// ---- VISUs/HMI_SenSimTest.TcVIS
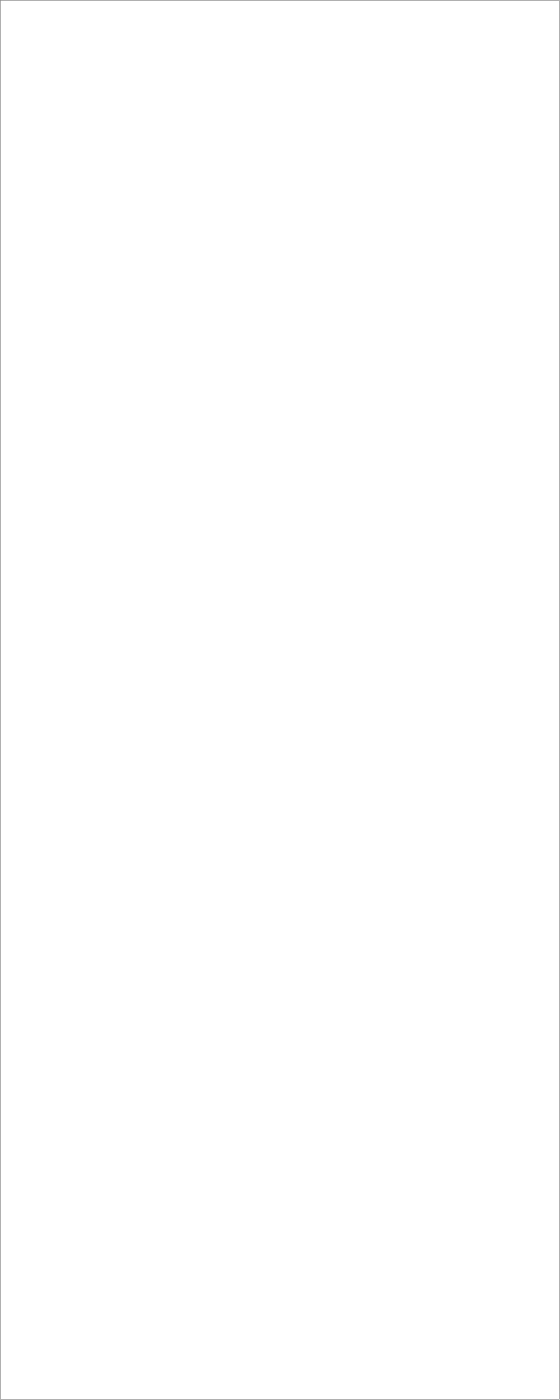
VISUALIZATION HMI_SenSimTest  // 801x2002
    Rectangle (7,175 430x823)
    Rectangle (260,175 176x823)
    Rectangle (7,875 429x23)
    Rectangle (7,741 429x23)
    Rectangle (7,174 429x23)
    Rectangle (6,16 669x143)
    Rectangle (6,17 669x32), "Manual Command Simulation From PLC"
    Checkbox (395,232 30x31), "Checkbox", tooltip "Enable Simulation", variable: stHMITIISenSimArray[iHMICbLevelSelection].bHMITIIByPassArray[1]
    ComboBoxInteger (295,235 100x25), tooltip "BackDoorSimulationMode", variable: arrTCMultiLevel[iHMICbLevelSelection].fbTCMultiLevelSeq.stMLBIO.ipAPPresentSensor, text list: 'BDList'
    RoundedRectangle (265,234 26x26), tooltip "VIO Status", colour toggle: arrTCMultiLevel[iHMICbLevelSelection].fbTCMultiLevelSeq.stMLVIO.ipAPPresentSensor
    Checkbox (263,201 164x31), "TIISen:VIOSim Override", variable: bHMIEnTIISenSimulation
    Checkbox (395,263 30x31), "Checkbox", tooltip "Enable Simulation", variable: stHMITIISenSimArray[iHMICbLevelSelection].bHMITIIByPassArray[2]
    ComboBoxInteger (295,267 100x25), tooltip "BackDoorSimulationMode", variable: arrTCMultiLevel[iHMICbLevelSelection].fbTCMultiLevelSeq.stMLBIO.ipAPPowerOn, text list: 'BDList'
    RoundedRectangle (265,265 26x26), tooltip "VIO Status", colour toggle: arrTCMultiLevel[iHMICbLevelSelection].fbTCMultiLevelSeq.stMLVIO.ipAPPowerOn
    Checkbox (395,294 30x31), "Checkbox", tooltip "Enable Simulation", variable: stHMITIISenSimArray[iHMICbLevelSelection].bHMITIIByPassArray[3]
    ComboBoxInteger (295,298 100x25), tooltip "BackDoorSimulationMode", variable: arrTCMultiLevel[iHMICbLevelSelection].fbTCMultiLevelSeq.stMLBIO.ipAPReady, text list: 'BDList'
    RoundedRectangle (265,296 26x26), tooltip "VIO Status", colour toggle: arrTCMultiLevel[iHMICbLevelSelection].fbTCMultiLevelSeq.stMLVIO.ipAPReady
    Checkbox (395,325 30x31), "Checkbox", tooltip "Enable Simulation", variable: stHMITIISenSimArray[iHMICbLevelSelection].bHMITIIByPassArray[4]
    ComboBoxInteger (295,328 100x25), tooltip "BackDoorSimulationMode", variable: arrTCMultiLevel[iHMICbLevelSelection].fbTCMultiLevelSeq.stMLBIO.ipHandlerSafeToEnterPLC, text list: 'BDList'
    RoundedRectangle (265,327 26x26), tooltip "VIO Status", colour toggle: arrTCMultiLevel[iHMICbLevelSelection].fbTCMultiLevelSeq.stMLVIO.ipHandlerSafeToEnterPLC
    Checkbox (395,356 30x31), "Checkbox", tooltip "Enable Simulation", variable: stHMITIISenSimArray[iHMICbLevelSelection].bHMITIIByPassArray[5]
    ComboBoxInteger (295,359 100x25), tooltip "BackDoorSimulationMode", variable: arrTCMultiLevel[iHMICbLevelSelection].fbTCMultiLevelSeq.stMLBIO.ipHandlerSafeToEnterHwr, text list: 'BDList'
    RoundedRectangle (265,358 26x26), tooltip "VIO Status", colour toggle: arrTCMultiLevel[iHMICbLevelSelection].fbTCMultiLevelSeq.stMLVIO.ipHandlerSafeToEnterHwr
    Checkbox (395,387 30x31), "Checkbox", tooltip "Enable Simulation", variable: stHMITIISenSimArray[iHMICbLevelSelection].bHMITIIByPassArray[6]
    ComboBoxInteger (295,390 100x25), tooltip "BackDoorSimulationMode", variable: arrTCMultiLevel[iHMICbLevelSelection].fbTCMultiLevelSeq.stMLBIO.ipCellFluidLeakage1, text list: 'BDList'
    RoundedRectangle (265,389 26x26), tooltip "VIO Status", colour toggle: arrTCMultiLevel[iHMICbLevelSelection].fbTCMultiLevelSeq.stMLVIO.ipCellFluidLeakage1
    Checkbox (395,418 30x31), "Checkbox", tooltip "Enable Simulation", variable: stHMITIISenSimArray[iHMICbLevelSelection].bHMITIIByPassArray[7]
    ComboBoxInteger (295,421 100x25), tooltip "BackDoorSimulationMode", variable: arrTCMultiLevel[iHMICbLevelSelection].fbTCMultiLevelSeq.stMLBIO.ipCellFluidLeakage2, text list: 'BDList'
    RoundedRectangle (265,420 26x26), tooltip "VIO Status", colour toggle: arrTCMultiLevel[iHMICbLevelSelection].fbTCMultiLevelSeq.stMLVIO.ipCellFluidLeakage2
    Checkbox (395,449 30x31), "Checkbox", tooltip "Enable Simulation", variable: stHMITIISenSimArray[iHMICbLevelSelection].bHMITIIByPassArray[8]
    ComboBoxInteger (295,452 100x25), tooltip "BackDoorSimulationMode", variable: arrTCMultiLevel[iHMICbLevelSelection].fbTCMultiLevelSeq.stMLBIO.ipCellGroundFault, text list: 'BDList'
    RoundedRectangle (265,451 26x26), tooltip "VIO Status", colour toggle: arrTCMultiLevel[iHMICbLevelSelection].fbTCMultiLevelSeq.stMLVIO.ipCellGroundFault
    Checkbox (395,480 30x31), "Checkbox", tooltip "Enable Simulation", variable: stHMITIISenSimArray[iHMICbLevelSelection].bHMITIIByPassArray[9]
    ComboBoxInteger (295,483 100x25), tooltip "BackDoorSimulationMode", variable: arrTCMultiLevel[iHMICbLevelSelection].fbTCMultiLevelSeq.stMLBIO.ipTesterPresent, text list: 'BDList'
    RoundedRectangle (265,482 26x26), tooltip "VIO Status", colour toggle: arrTCMultiLevel[iHMICbLevelSelection].fbTCMultiLevelSeq.stMLVIO.ipTesterPresent
    Checkbox (395,511 30x31), "Checkbox", tooltip "Enable Simulation", variable: stHMITIISenSimArray[iHMICbLevelSelection].bHMITIIByPassArray[10]
    ComboBoxInteger (295,514 100x25), tooltip "BackDoorSimulationMode", variable: arrTCMultiLevel[iHMICbLevelSelection].fbTCMultiLevelSeq.stMLBIO.ipTesterPowerOn, text list: 'BDList'
    RoundedRectangle (265,513 26x26), tooltip "VIO Status", colour toggle: arrTCMultiLevel[iHMICbLevelSelection].fbTCMultiLevelSeq.stMLVIO.ipTesterPowerOn
    Checkbox (395,542 30x31), "Checkbox", tooltip "Enable Simulation", variable: stHMITIISenSimArray[iHMICbLevelSelection].bHMITIIByPassArray[11]
    ComboBoxInteger (295,545 100x25), tooltip "BackDoorSimulationMode", variable: arrTCMultiLevel[iHMICbLevelSelection].fbTCMultiLevelSeq.stMLBIO.ipTesterReady, text list: 'BDList'
    RoundedRectangle (265,544 26x26), tooltip "VIO Status", colour toggle: arrTCMultiLevel[iHMICbLevelSelection].fbTCMultiLevelSeq.stMLVIO.ipTesterReady
    Checkbox (395,573 30x31), "Checkbox", tooltip "Enable Simulation", variable: stHMITIISenSimArray[iHMICbLevelSelection].bHMITIIByPassArray[12]
    ComboBoxInteger (295,576 100x25), tooltip "BackDoorSimulationMode", variable: arrTCMultiLevel[iHMICbLevelSelection].fbTCMultiLevelSeq.stMLBIO.ipTCCellDoorClosed, text list: 'BDList'
    RoundedRectangle (265,575 26x26), tooltip "VIO Status", colour toggle: arrTCMultiLevel[iHMICbLevelSelection].fbTCMultiLevelSeq.stMLVIO.ipTCCellDoorClosed
    Checkbox (395,604 30x31), "Checkbox", tooltip "Enable Simulation", variable: stHMITIISenSimArray[iHMICbLevelSelection].bHMITIIByPassArray[13]
    ComboBoxInteger (295,607 100x25), tooltip "BackDoorSimulationMode", variable: arrTCMultiLevel[iHMICbLevelSelection].fbTCMultiLevelSeq.stMLBIO.ipTesterLatchesClosed, text list: 'BDList'
    RoundedRectangle (265,606 26x26), tooltip "VIO Status", colour toggle: arrTCMultiLevel[iHMICbLevelSelection].fbTCMultiLevelSeq.stMLVIO.ipTesterLatchesClosed
    Checkbox (395,635 30x31), "Checkbox", tooltip "Enable Simulation", variable: stHMITIISenSimArray[iHMICbLevelSelection].bHMITIIByPassArray[14]
    ComboBoxInteger (295,638 100x25), tooltip "BackDoorSimulationMode", variable: arrTCMultiLevel[iHMICbLevelSelection].fbTCMultiLevelSeq.stMLBIO.ipTIUPresent, text list: 'BDList'
    RoundedRectangle (265,637 26x26), tooltip "VIO Status", colour toggle: arrTCMultiLevel[iHMICbLevelSelection].fbTCMultiLevelSeq.stMLVIO.ipTIUPresent
    Checkbox (395,666 30x31), "Checkbox", tooltip "Enable Simulation"
    ComboBoxInteger (295,669 100x25), tooltip "BackDoorSimulationMode", variable: arrTCMultiLevel[iHMICbLevelSelection].fbTCMultiLevelSeq.stMLBIO.ipAPPresentSensor, text list: 'BDList'
    RoundedRectangle (265,668 26x26), tooltip "VIO Status"
    Checkbox (395,697 30x31), "Checkbox", tooltip "Enable Simulation"
    ComboBoxInteger (295,700 100x25), tooltip "BackDoorSimulationMode", variable: arrTCMultiLevel[iHMICbLevelSelection].fbTCMultiLevelSeq.stMLBIO.ipAPPresentSensor, text list: 'BDList'
    RoundedRectangle (265,699 26x26), tooltip "VIO Status"
    RoundedRectangle (69,234 165x25), "01)_AP_PresentSensor*"
    Checkbox (12,232 30x31), "Checkbox", tooltip "Enable Simulation", variable: stHMITIIByPassArray[iHMICbLevelSelection].bHMITIIByPassArray[1]
    RoundedRectangle (69,265 165x25), "02)_AP_PowerOn*"
    Checkbox (12,263 30x31), "Checkbox", tooltip "Enable Simulation", variable: stHMITIIByPassArray[iHMICbLevelSelection].bHMITIIByPassArray[2]
    RoundedRectangle (69,296 165x25), "03)_AP_Ready"
    Checkbox (12,294 30x31), "Checkbox", tooltip "Enable Simulation", variable: stHMITIIByPassArray[iHMICbLevelSelection].bHMITIIByPassArray[3]
    RoundedRectangle (69,327 165x25), "04)_AP_DeactuatedPLC`*`"
    Checkbox (12,325 30x31), "Checkbox", tooltip "Enable Simulation", variable: stHMITIIByPassArray[iHMICbLevelSelection].bHMITIIByPassArray[4]
    RoundedRectangle (69,358 165x25), "05)_AP_DeactuatedHwr`*`"
    Checkbox (12,356 30x31), "Checkbox", tooltip "Enable Simulation", variable: stHMITIIByPassArray[iHMICbLevelSelection].bHMITIIByPassArray[5]
    RoundedRectangle (69,389 165x25), "06)_CellFluidLeakage1"
    Checkbox (12,387 30x31), "Checkbox", tooltip "Enable Simulation", variable: stHMITIIByPassArray[iHMICbLevelSelection].bHMITIIByPassArray[6]
    RoundedRectangle (69,420 165x25), "07)_CellFluidLeakage2"
    Checkbox (12,418 30x31), "Checkbox", tooltip "Enable Simulation", variable: stHMITIIByPassArray[iHMICbLevelSelection].bHMITIIByPassArray[7]
    RoundedRectangle (69,451 165x25), "08)_CellGroundFault"
    Checkbox (12,449 30x31), "Checkbox", tooltip "Enable Simulation", variable: stHMITIIByPassArray[iHMICbLevelSelection].bHMITIIByPassArray[8]
    RoundedRectangle (69,482 165x25), "09)_TesterPresent**"
    Checkbox (12,480 30x31), "Checkbox", tooltip "Enable Simulation", variable: stHMITIIByPassArray[iHMICbLevelSelection].bHMITIIByPassArray[9]
    RoundedRectangle (69,513 165x25), "10)_TesterPowerOn**"
    Checkbox (12,511 30x31), "Checkbox", tooltip "Enable Simulation", variable: stHMITIIByPassArray[iHMICbLevelSelection].bHMITIIByPassArray[10]
    RoundedRectangle (69,544 165x25), "11)_TesterReady"
    Checkbox (12,542 30x31), "Checkbox", tooltip "Enable Simulation", variable: stHMITIIByPassArray[iHMICbLevelSelection].bHMITIIByPassArray[11]
    RoundedRectangle (69,575 165x25), "12)_TCCellDoorClosed"
    Checkbox (12,573 30x31), "Checkbox", tooltip "Enable Simulation", variable: stHMITIIByPassArray[iHMICbLevelSelection].bHMITIIByPassArray[12]
    RoundedRectangle (69,606 165x25), "13)_TesterLatchesClosed**"
    Checkbox (12,604 30x31), "Checkbox", tooltip "Enable Simulation", variable: stHMITIIByPassArray[iHMICbLevelSelection].bHMITIIByPassArray[13]
    RoundedRectangle (69,637 165x25), "14)_TIUPresent"
    Checkbox (12,635 30x31), "Checkbox", tooltip "Enable Simulation", variable: stHMITIIByPassArray[iHMICbLevelSelection].bHMITIIByPassArray[14]
    RoundedRectangle (69,668 165x25)
    Checkbox (12,666 30x31), "Checkbox", tooltip "Enable Simulation"
    RoundedRectangle (69,699 165x25)
    Checkbox (12,697 30x31), "Checkbox", tooltip "Enable Simulation"
    Checkbox (12,202 227x31), "TII Alarm Enable Override", variable: bHMITIIBypass
    Checkbox (629,331 30x31), "Checkbox", tooltip "Enable Simulation", variable: stHMIBtnSimArray[iHMICbLevelSelection].bHMITIIByPassArray[1]
    ComboBoxInteger (483,334 140x25), tooltip "BackDoorSimulationMode", variable: arrTCMultiLevel[iHMICbLevelSelection].fbTCMultiLevelSeq.stMLBIO.ipDrawerMaintenanceModeBtn, text list: 'BDList'
    RoundedRectangle (453,333 26x26), tooltip "VIO Status", colour toggle: arrTCMultiLevel[iHMICbLevelSelection].fbTCMultiLevelSeq.stMLVIO.ipDrawerMaintenanceModeBtn
    Checkbox (629,362 30x31), "Checkbox", tooltip "Enable Simulation", variable: stHMIBtnSimArray[iHMICbLevelSelection].bHMITIIByPassArray[2]
    ComboBoxInteger (483,366 140x25), tooltip "BackDoorSimulationMode", variable: arrTCMultiLevel[iHMICbLevelSelection].fbTCMultiLevelSeq.stMLBIO.ipTCCellAbortFlowBtn, text list: 'BDList'
    RoundedRectangle (453,364 26x26), tooltip "VIO Status", colour toggle: arrTCMultiLevel[iHMICbLevelSelection].fbTCMultiLevelSeq.stMLVIO.ipTCCellAbortFlowBtn
    Checkbox (629,393 30x31), "Checkbox", tooltip "Enable Simulation", variable: stHMIBtnSimArray[iHMICbLevelSelection].bHMITIIByPassArray[3]
    ComboBoxInteger (483,397 140x25), tooltip "BackDoorSimulationMode", variable: arrTCMultiLevel[iHMICbLevelSelection].fbTCMultiLevelSeq.stMLBIO.ipTCCellDoorOpenReqBtn, text list: 'BDList'
    RoundedRectangle (453,395 26x26), tooltip "VIO Status", colour toggle: arrTCMultiLevel[iHMICbLevelSelection].fbTCMultiLevelSeq.stMLVIO.ipTCCellDoorOpenReqBtn
    Checkbox (452,300 157x31), "Btn VIO Sim Override", variable: bHMIBtnSimulation
    Checkbox (454,427 150x30), "AutoRsetEvntTrigger", variable: bHMIRsetEvntTriggerOnProductionMode
    RoundedRectangle (41,234 26x26), tooltip "VIO Status", colour toggle: ALMTC.Level[iHMICbLevelSelection].AlarmID[1]
    RoundedRectangle (41,265 26x26), tooltip "VIO Status", colour toggle: ALMTC.Level[iHMICbLevelSelection].AlarmID[2]
    RoundedRectangle (41,296 26x26), tooltip "VIO Status", colour toggle: ALMTC.Level[iHMICbLevelSelection].AlarmID[3]
    RoundedRectangle (41,327 26x26), tooltip "VIO Status", colour toggle: ALMTC.Level[iHMICbLevelSelection].AlarmID[4]
    RoundedRectangle (41,358 26x26), tooltip "VIO Status", colour toggle: ALMTC.Level[iHMICbLevelSelection].AlarmID[5]
    RoundedRectangle (41,389 26x26), tooltip "VIO Status", colour toggle: ALMTC.Level[iHMICbLevelSelection].AlarmID[6]
    RoundedRectangle (41,420 26x26), tooltip "VIO Status", colour toggle: ALMTC.Level[iHMICbLevelSelection].AlarmID[7]
    RoundedRectangle (41,451 26x26), tooltip "VIO Status", colour toggle: ALMTC.Level[iHMICbLevelSelection].AlarmID[8]
    RoundedRectangle (41,482 26x26), tooltip "VIO Status", colour toggle: ALMTC.Level[iHMICbLevelSelection].AlarmID[9]
    RoundedRectangle (41,513 26x26), tooltip "VIO Status", colour toggle: ALMTC.Level[iHMICbLevelSelection].AlarmID[10]
    RoundedRectangle (41,544 26x26), tooltip "VIO Status", colour toggle: ALMTC.Level[iHMICbLevelSelection].AlarmID[11]
    RoundedRectangle (41,575 26x26), tooltip "VIO Status", colour toggle: ALMTC.Level[iHMICbLevelSelection].AlarmID[12]
    RoundedRectangle (41,606 26x26), tooltip "VIO Status", colour toggle: ALMTC.Level[iHMICbLevelSelection].AlarmID[13]
    RoundedRectangle (41,637 26x26), tooltip "VIO Status", colour toggle: ALMTC.Level[iHMICbLevelSelection].AlarmID[14]
    RoundedRectangle (41,668 26x26), tooltip "VIO Status"
    RoundedRectangle (41,699 26x26), tooltip "VIO Status"
    Checkbox (394,766 30x31), "Checkbox", tooltip "Enable Simulation", variable: bHMIColSenSimArray[1]
    ComboBoxInteger (294,769 100x25), tooltip "BackDoorSimulationMode", variable: fbTCColumn.stTCColumnBIO.ipColumnFluid_PCW_Leakage, text list: 'BDList'
    RoundedRectangle (264,768 26x26), tooltip "VIO Status", colour toggle: fbTCColumn.stTCColumnVIO.ipColumnFluid_PCW_Leakage
    Checkbox (394,797 30x31), "Checkbox", tooltip "Enable Simulation", variable: bHMIColSenSimArray[2]
    ComboBoxInteger (294,800 100x25), tooltip "BackDoorSimulationMode", variable: fbTCColumn.stTCColumnBIO.ipAllTCDrawerRetractedinCell, text list: 'BDList'
    RoundedRectangle (264,799 26x26), tooltip "VIO Status", colour toggle: fbTCColumn.stTCColumnVIO.ipAllTCDrawerRetractedinCell
    Checkbox (394,828 30x31), "Checkbox", tooltip "Enable Simulation", variable: bHMIColSenSimArray[3]
    ComboBoxInteger (294,831 100x25), tooltip "BackDoorSimulationMode", variable: fbTCColumn.stTCColumnBIO.ipSystem_ipColumnGroundFault, text list: 'BDList'
    RoundedRectangle (264,830 26x26), tooltip "VIO Status", colour toggle: fbTCColumn.stTCColumnVIO.ipSystem_ipColumnGroundFault
    RoundedRectangle (71,769 162x25), "1)_Col_Leakage"
    Checkbox (12,767 30x31), "Checkbox", tooltip "Enable Simulation", variable: arrHMISysAlmByPass[1]
    RoundedRectangle (71,800 162x25), "2)_All_Dwr_Ret"
    Checkbox (12,799 30x31), "Checkbox", tooltip "Enable Simulation", variable: arrHMISysAlmByPass[2]
    RoundedRectangle (71,831 162x25), "3)_Col_Grd"
    Checkbox (12,830 30x31), "Checkbox", tooltip "Enable Simulation", variable: arrHMISysAlmByPass[3]
    RoundedRectangle (42,769 26x26), tooltip "VIO Status", colour toggle: ALMTC.Common.AlarmID[1]
    RoundedRectangle (42,800 26x26), tooltip "VIO Status", colour toggle: ALMTC.Common.AlarmID[2]
    RoundedRectangle (42,831 26x26), tooltip "VIO Status", colour toggle: ALMTC.Common.AlarmID[3]
    RoundedRectangle (476,233 181x25), "ButtonModeConditionSimulation"
        toggle arrHMIBtnSolidOn_Condition[iHMICbLevelSelection,iHMIBtnType]
    RoundedRectangle (449,233 25x25), colour toggle: arrHMIBtnSolidOn_Condition[iHMICbLevelSelection,iHMIBtnType]
    ComboBoxInteger (451,266 208x25), tooltip "BackDoorSimulationMode", variable: iHMIBtnType, text list: 'BtnTxtList'
    ComboBoxInteger (106,71 188x30), variable: iHMICbCmdSelection, text list: 'CmdTxtList'
    ComboBoxInteger (14,71 89x30), variable: iHMICbLevelSelection, text list: 'LevelTxtList'
    Button (12,108 281x45), "Test Command"
        tap TestManually.bTestCommand
    ComboBoxInteger (306,73 276x25), variable: TestManually.iAlarmCode, text list: 'AlarmTxtList'
    Checkbox (586,68 37x30), variable: bHMIResetAllAlarm
    Label (616,68 183x30), "Reset All"
    Label (304,50 215x30), "Individual Alarm ID:"
    Button (302,111 281x42), "Init All Level"
        tap TestManually.bInitialiseAll
    Checkbox (397,900 30x31), "Checkbox", tooltip "Enable Simulation", variable: stDebugStation.fbDBStnSeq.bTIISenSimArray[1]
    ComboBoxInteger (297,903 100x25), tooltip "BackDoorSimulationMode", variable: stDebugStation.fbDBStnSeq.stDebugStationBIO.ipDBStnAPPresentSensor, text list: 'BDList'
    RoundedRectangle (267,902 26x26), tooltip "VIO Status", colour toggle: stDebugStation.fbDBStnSeq.stDebugStationVIO.ipDBStnAPPresentSensor
    Checkbox (397,931 30x31), "Checkbox", tooltip "Enable Simulation", variable: stDebugStation.fbDBStnSeq.bTIISenSimArray[2]
    ComboBoxInteger (297,935 100x25), tooltip "BackDoorSimulationMode", variable: stDebugStation.fbDBStnSeq.stDebugStationBIO.ipDBStnAPPowerOn, text list: 'BDList'
    RoundedRectangle (267,933 26x26), tooltip "VIO Status", colour toggle: stDebugStation.fbDBStnSeq.stDebugStationVIO.ipDBStnAPPowerOn
    Checkbox (397,962 30x31), "Checkbox", tooltip "Enable Simulation", variable: stDebugStation.fbDBStnSeq.bTIISenSimArray[3]
    ComboBoxInteger (297,966 100x25), tooltip "BackDoorSimulationMode", variable: stDebugStation.fbDBStnSeq.stDebugStationBIO.ipDBStnAPReady, text list: 'BDList'
    RoundedRectangle (267,964 26x26), tooltip "VIO Status", colour toggle: stDebugStation.fbDBStnSeq.stDebugStationVIO.ipDBStnAPReady
    RoundedRectangle (71,902 165x25), "01)_AP_PresentSensor"
    Checkbox (14,900 30x31), "Checkbox", tooltip "Enable Simulation", variable: stHMITIIByPassArray[iHMICbLevelSelection].bHMITIIByPassArray[1]
    RoundedRectangle (71,933 165x25), "02)_AP_PowerOn"
    Checkbox (14,931 30x31), "Checkbox", tooltip "Enable Simulation", variable: stHMITIIByPassArray[iHMICbLevelSelection].bHMITIIByPassArray[2]
    RoundedRectangle (71,964 165x25), "03)_AP_Ready"
    Checkbox (14,962 30x31), "Checkbox", tooltip "Enable Simulation", variable: stHMITIIByPassArray[iHMICbLevelSelection].bHMITIIByPassArray[3]
    RoundedRectangle (43,902 26x26), tooltip "VIO Status", colour toggle: ALMTC.Level[iHMICbLevelSelection].AlarmID[1]
    RoundedRectangle (43,933 26x26), tooltip "VIO Status", colour toggle: ALMTC.Level[iHMICbLevelSelection].AlarmID[2]
    RoundedRectangle (43,964 26x26), tooltip "VIO Status", colour toggle: ALMTC.Level[iHMICbLevelSelection].AlarmID[3]
    Label (20,871 183x30), "DEBUG STATION"
    Label (15,171 183x30), "CELL STACK"
    Label (20,740 183x30), "COLUMN"
    Group (452,468 225x262)
        Rectangle (0,0 215x259)
        Rectangle (0,237 215x22)
        RoundedRectangle (7,206 60x26), "Level[1]", tooltip "VIO Status", colour toggle: TC_ModuleState[1].Tester = E_State.eEnabled
        RoundedRectangle (7,177 60x26), "Level[2]", tooltip "VIO Status", colour toggle: TC_ModuleState[2].Tester= E_State.eEnabled
        RoundedRectangle (7,148 60x26), "Level[3]", tooltip "VIO Status", colour toggle: TC_ModuleState[3].Tester = E_State.eEnabled
        RoundedRectangle (7,119 60x26), "Level[4]", tooltip "VIO Status", colour toggle: TC_ModuleState[4].Tester = E_State.eEnabled
        RoundedRectangle (7,90 60x26), "Level[5]", tooltip "VIO Status", colour toggle: TC_ModuleState[5].Tester = E_State.eEnabled
        RoundedRectangle (7,61 60x26), "Level[6]", tooltip "VIO Status", colour toggle: TC_ModuleState[6].Tester = E_State.eEnabled
        Label (6,32 61x30), "Tester"
        RoundedRectangle (149,206 60x26), "Level[1]", tooltip "VIO Status", colour toggle: TC_ModuleState[1].TCSite[1].TIERII = E_State.eEnabled
        RoundedRectangle (149,177 60x26), "Level[2]", tooltip "VIO Status", colour toggle: TC_ModuleState[2].TCSite[1].TIERII = E_State.eEnabled
        RoundedRectangle (149,148 60x26), "Level[3]", tooltip "VIO Status", colour toggle: TC_ModuleState[3].TCSite[1].TIERII = E_State.eEnabled
        RoundedRectangle (149,119 60x26), "Level[4]", tooltip "VIO Status", colour toggle: TC_ModuleState[4].TCSite[1].TIERII = E_State.eEnabled
        RoundedRectangle (149,90 60x26), "Level[5]", tooltip "VIO Status", colour toggle: TC_ModuleState[5].TCSite[1].TIERII = E_State.eEnabled
        RoundedRectangle (149,61 60x26), "Level[6]", tooltip "VIO Status", colour toggle: TC_ModuleState[6].TCSite[1].TIERII = E_State.eEnabled
        Label (162,32 32x30), "TII"
        RoundedRectangle (78,207 60x26), "Level[1]", tooltip "VIO Status", colour toggle: TC_ModuleState[1].TCSite[1].TCU = E_State.eEnabled
        RoundedRectangle (78,178 60x26), "Level[2]", tooltip "VIO Status", colour toggle: TC_ModuleState[2].TCSite[1].TCU= E_State.eEnabled
        RoundedRectangle (78,149 60x26), "Level[3]", tooltip "VIO Status", colour toggle: TC_ModuleState[3].TCSite[1].TCU = E_State.eEnabled
        RoundedRectangle (78,120 60x26), "Level[4]", tooltip "VIO Status", colour toggle: TC_ModuleState[4].TCSite[1].TCU = E_State.eEnabled
        RoundedRectangle (78,91 60x26), "Level[5]", tooltip "VIO Status", colour toggle: TC_ModuleState[5].TCSite[1].TCU = E_State.eEnabled
        RoundedRectangle (78,62 60x26), "Level[6]", tooltip "VIO Status", colour toggle: TC_ModuleState[6].TCSite[1].TCU = E_State.eEnabled
        Label (87,33 43x30), "TCU"
        Label (12,232 213x30), "Green: Enable , Gray: Disable"
        Rectangle (0,1 215x32), "Enable/ Disable Status"
    Rectangle (7,1009 430x271)
    Rectangle (7,1010 429x32), "Manual Command Simulation From PLC"
    Label (9,1073 153x30), "AP240PwrCheckDelay(ms)"
    Textfield (162,1073 103x30), "%i", text variable: APPwrOnChkDelay, input disabled if: TRUE
        OnMouseClick: write the text variable via Default
    Button (383,1074 50x30), "Write", input disabled if: NOT (iAPPwrOnChkDelay>=0)
        tap BtnSetAPPwrOnChkDelay
    Label (165,1047 78x30), "Current Value"
    Label (276,1046 84x30), "Value To Write"
    Textfield (272,1073 103x30), "%i", text variable: iAPPwrOnChkDelay
        OnMouseClick: write the text variable via Default
    Label (8,1109 154x30), "Tst240PwrCheckDelay(ms)"
    Textfield (162,1109 103x30), "%i", text variable: TstPwrOnChkDelay, input disabled if: TRUE
        OnMouseClick: write the text variable via Default
    Button (383,1110 50x30), "Write", input disabled if: NOT (iTstPwrOnChkDelay>=0)
        tap BtnSetTstPwrOnChkDelay
    Textfield (272,1109 103x30), "%i", text variable: iTstPwrOnChkDelay
        OnMouseClick: write the text variable via Default
    Label (9,1150 153x30), "APReadyCheckDelay(ms)"
    Textfield (162,1150 103x30), "%i", text variable: APPwrOnChkDelay, input disabled if: TRUE
        OnMouseClick: write the text variable via Default
    Button (383,1151 50x30), "Write", input disabled if: NOT (iAPPwrOnChkDelay>=0)
        tap BtnSetAPPwrOnChkDelay
    Textfield (272,1150 103x30), "%i", text variable: iAPPwrOnChkDelay
        OnMouseClick: write the text variable via Default
    Label (8,1186 154x30), "TstReadyCheckDelay(ms)"
    Textfield (162,1186 103x30), "%i", text variable: TstPwrOnChkDelay, input disabled if: TRUE
        OnMouseClick: write the text variable via Default
    Button (383,1187 50x30), "Write", input disabled if: NOT (iTstPwrOnChkDelay>=0)
        tap BtnSetTstPwrOnChkDelay
    Textfield (272,1186 103x30), "%i", text variable: iTstPwrOnChkDelay
        OnMouseClick: write the text variable via Default
    Rectangle (0,0 792x2000), invisible if: bEnableManualCommandTest1 AND bEnableManualCommandTest2
END_VISUALIZATION

// ---- VISUs/HMI_All_Level.TcVIS
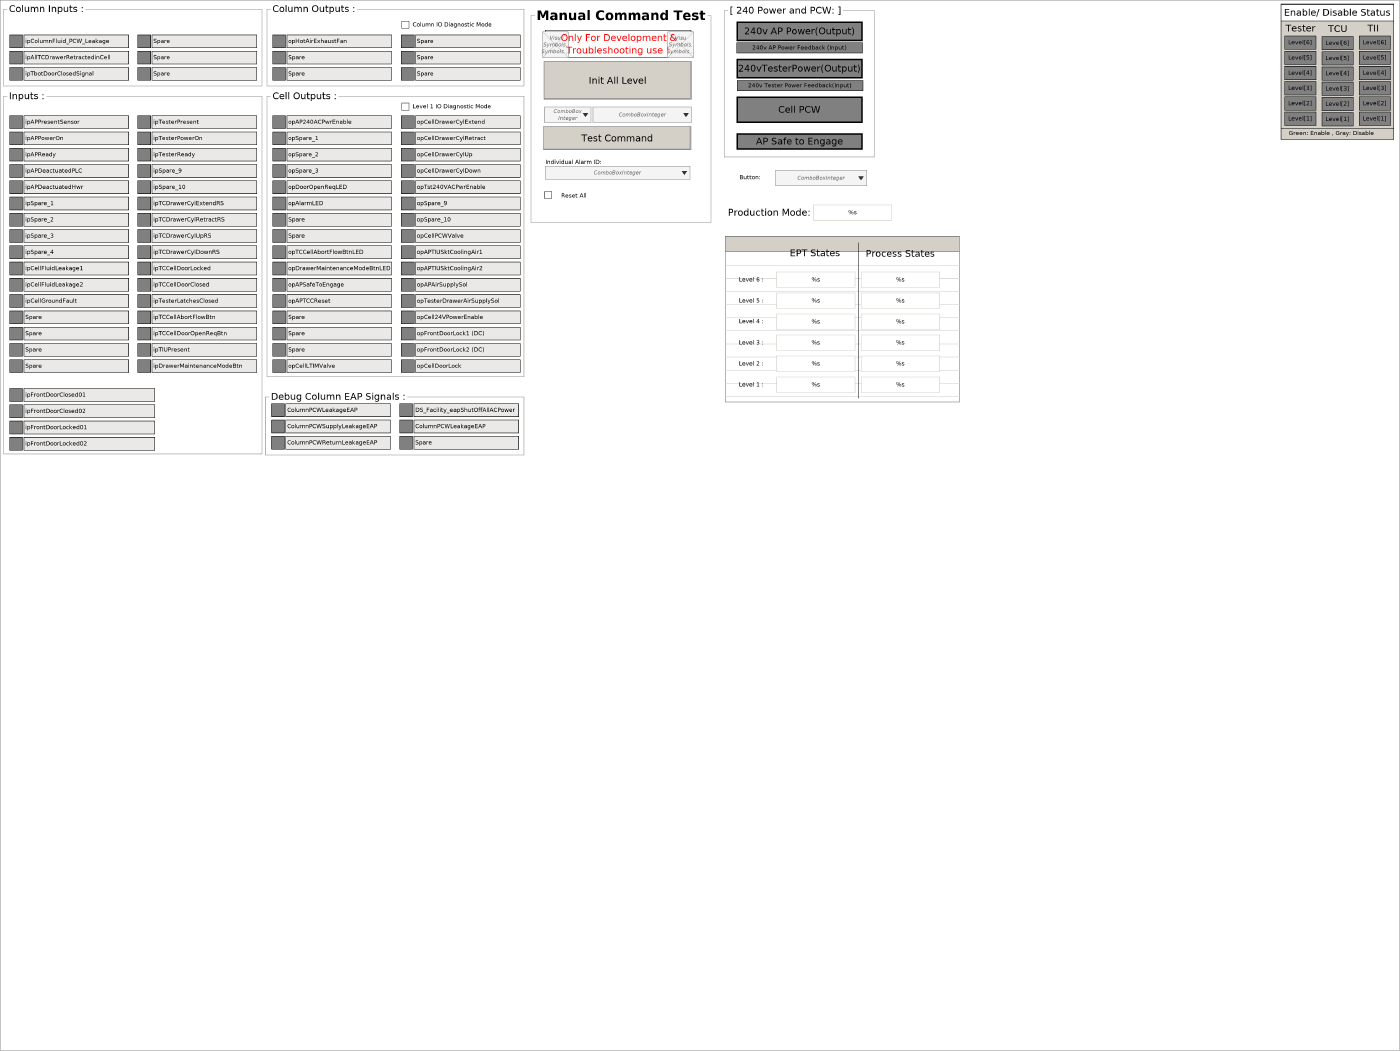
VISUALIZATION HMI_All_Level  // 2667x2003
    Table (1381,450 447x316)
    GroupBox (1379,12 287x287), "[ 240 Power and PCW: ]"
        RoundedRectangle (24,69 240x20), "240v AP Power Feedback (Input)", colour toggle: arrTCMultiLevel[iHMICbLevelSelection].fbTCMultiLevelSeq.stMLDIO.ipAPPowerOn
        RoundedRectangle (25,141 240x20), "240v Tester Power Feedback(Input)", colour toggle: arrTCMultiLevel[iHMICbLevelSelection].fbTCMultiLevelSeq.stMLDIO.ipTesterPowerOn
        RoundedRectangle (24,242 240x31), "AP Safe to Engage", colour toggle: arrTCMultiLevel[iHMICbLevelSelection].fbTCMultiLevelSeq.stMLDIO.opAPSafeToEngage
    GroupBox (6,175 493x690), "Inputs :"
        RoundedRectangle (12,510 25x25)
        RoundedRectangle (256,510 25x25), colour toggle: arrTCMultiLevel[iHMICbLevelSelection].fbTCMultiLevelSeq.stMLDIO.ipDrawerMaintenanceModeBtn
    GroupBox (508,175 490x543), "Cell Outputs :"
        RoundedRectangle (283,45 200x25), "opCellDrawerCylExtend"
            toggle arrTCMultiLevel[iHMICbLevelSelection].fbTCMultiLevelSeq.stMLDIO.opCellDrawerCylExtend
        RoundedRectangle (38,479 200x25), "Spare"
    RoundedRectangle (546,220 200x25), "opAP240ACPwrEnable"
        toggle arrTCMultiLevel[iHMICbLevelSelection].fbTCMultiLevelSeq.stMLDIO.opAP240ACPwrEnable
    RoundedRectangle (546,251 200x25), "opSpare_1"
        toggle arrTCMultiLevel[iHMICbLevelSelection].fbTCMultiLevelSeq.stMLDIO.opSpare_1
    RoundedRectangle (546,282 200x25), "opSpare_2"
        toggle arrTCMultiLevel[iHMICbLevelSelection].fbTCMultiLevelSeq.stMLDIO.opSpare_2
    RoundedRectangle (546,313 200x25), "opSpare_3"
        toggle arrTCMultiLevel[iHMICbLevelSelection].fbTCMultiLevelSeq.stMLDIO.opSpare_3
    RoundedRectangle (546,344 200x25), "opDoorOpenReqLED"
        toggle arrTCMultiLevel[iHMICbLevelSelection].fbTCMultiLevelSeq.stMLDIO.opDoorOpenReqLED
    RoundedRectangle (546,375 200x25), "opAlarmLED"
        toggle arrTCMultiLevel[iHMICbLevelSelection].fbTCMultiLevelSeq.stMLDIO.opAlarmLED
    RoundedRectangle (546,406 200x25), "Spare"
    RoundedRectangle (546,437 200x25), "Spare"
    RoundedRectangle (546,468 200x25), "opTCCellAbortFlowBtnLED"
        toggle arrTCMultiLevel[iHMICbLevelSelection].fbTCMultiLevelSeq.stMLDIO.opTCCellAbortFlowBtnLED
    RoundedRectangle (546,499 200x25), "opDrawerMaintenanceModeBtnLED"
        toggle arrTCMultiLevel[iHMICbLevelSelection].fbTCMultiLevelSeq.stMLDIO.opDrawerMaintenanceModeBtnLED
    RoundedRectangle (546,530 200x25), "opAPSafeToEngage"
        toggle arrTCMultiLevel[iHMICbLevelSelection].fbTCMultiLevelSeq.stMLDIO.opAPSafeToEngage
    RoundedRectangle (546,561 200x25), "opAPTCCReset"
        toggle arrTCMultiLevel[iHMICbLevelSelection].fbTCMultiLevelSeq.stMLDIO.opAPTCCReset
    RoundedRectangle (546,592 200x25), "Spare"
    RoundedRectangle (546,623 200x25), "Spare"
    RoundedRectangle (791,654 200x25), "opFrontDoorLock2 (DC)"
        toggle arrTCMultiLevel[iHMICbLevelSelection].fbTCMultiLevelSeq.stMLDIO.opCellTBOtSideDoorClosed2
    RoundedRectangle (546,685 200x25), "opCellLTIMValve"
        toggle arrTCMultiLevel[iHMICbLevelSelection].fbTCMultiLevelSeq.stMLDIO.opCellLTIMValve
    RoundedRectangle (519,220 25x25), colour toggle: arrTCMultiLevel[iHMICbLevelSelection].fbTCMultiLevelSeq.stMLDIO.opAP240ACPwrEnable
    RoundedRectangle (519,251 25x25), colour toggle: arrTCMultiLevel[iHMICbLevelSelection].fbTCMultiLevelSeq.stMLDIO.opSpare_1
    RoundedRectangle (519,282 25x25), colour toggle: arrTCMultiLevel[iHMICbLevelSelection].fbTCMultiLevelSeq.stMLDIO.opSpare_2
    RoundedRectangle (519,313 25x25), colour toggle: arrTCMultiLevel[iHMICbLevelSelection].fbTCMultiLevelSeq.stMLDIO.opSpare_3
    RoundedRectangle (519,344 25x25), colour toggle: arrTCMultiLevel[iHMICbLevelSelection].fbTCMultiLevelSeq.stMLDIO.opDoorOpenReqLED
    RoundedRectangle (519,375 25x25), colour toggle: arrTCMultiLevel[iHMICbLevelSelection].fbTCMultiLevelSeq.stMLDIO.opAlarmLED
    RoundedRectangle (519,406 25x25)
    RoundedRectangle (519,437 25x25)
    RoundedRectangle (519,468 25x25), colour toggle: arrTCMultiLevel[iHMICbLevelSelection].fbTCMultiLevelSeq.stMLDIO.opTCCellAbortFlowBtnLED
    RoundedRectangle (519,499 25x25), colour toggle: arrTCMultiLevel[iHMICbLevelSelection].fbTCMultiLevelSeq.stMLDIO.opDrawerMaintenanceModeBtnLED
    RoundedRectangle (519,530 25x25), colour toggle: arrTCMultiLevel[iHMICbLevelSelection].fbTCMultiLevelSeq.stMLDIO.opAPSafeToEngage
    RoundedRectangle (519,561 25x25), colour toggle: arrTCMultiLevel[iHMICbLevelSelection].fbTCMultiLevelSeq.stMLDIO.opAPTCCReset
    RoundedRectangle (519,592 25x25)
    RoundedRectangle (519,623 25x25)
    RoundedRectangle (519,654 25x25)
    RoundedRectangle (519,685 25x25), colour toggle: arrTCMultiLevel[iHMICbLevelSelection].fbTCMultiLevelSeq.stMLDIO.opCellLTIMValve
    RoundedRectangle (45,220 200x25), "ipAPPresentSensor"
    RoundedRectangle (45,251 200x25), "ipAPPowerOn"
    RoundedRectangle (45,282 200x25), "ipAPReady"
    RoundedRectangle (45,313 200x25), "ipAPDeactuatedPLC"
    RoundedRectangle (45,344 200x25), "ipAPDeactuatedHwr"
    RoundedRectangle (45,375 200x25), "ipSpare_1"
    RoundedRectangle (45,406 200x25), "ipSpare_2"
    RoundedRectangle (45,437 200x25), "ipSpare_3"
    RoundedRectangle (45,468 200x25), "ipSpare_4"
    RoundedRectangle (45,499 200x25), "ipCellFluidLeakage1"
    RoundedRectangle (45,530 200x25), "ipCellFluidLeakage2"
    RoundedRectangle (45,561 200x25), "ipCellGroundFault"
    RoundedRectangle (45,592 200x25), "Spare"
    RoundedRectangle (45,623 200x25), "Spare"
    RoundedRectangle (45,654 200x25), "Spare"
    RoundedRectangle (45,685 200x25), "Spare"
    RoundedRectangle (18,220 25x25), colour toggle: arrTCMultiLevel[iHMICbLevelSelection].fbTCMultiLevelSeq.stMLDIO.ipAPPresentSensor
    RoundedRectangle (18,251 25x25), colour toggle: arrTCMultiLevel[iHMICbLevelSelection].fbTCMultiLevelSeq.stMLDIO.ipAPPowerOn
    RoundedRectangle (18,282 25x25), colour toggle: arrTCMultiLevel[iHMICbLevelSelection].fbTCMultiLevelSeq.stMLDIO.ipAPReady
    RoundedRectangle (18,313 25x25), colour toggle: arrTCMultiLevel[iHMICbLevelSelection].fbTCMultiLevelSeq.stMLDIO.ipHandlerSafeToEnterPLC
    RoundedRectangle (18,344 25x25), colour toggle: arrTCMultiLevel[iHMICbLevelSelection].fbTCMultiLevelSeq.stMLDIO.ipHandlerSafeToEnterHwr
    RoundedRectangle (18,375 25x25), colour toggle: arrTCMultiLevel[iHMICbLevelSelection].fbTCMultiLevelSeq.stMLDIO.ipSpare_1
    RoundedRectangle (18,406 25x25), colour toggle: arrTCMultiLevel[iHMICbLevelSelection].fbTCMultiLevelSeq.stMLDIO.ipSpare_2
    RoundedRectangle (18,437 25x25), colour toggle: arrTCMultiLevel[iHMICbLevelSelection].fbTCMultiLevelSeq.stMLDIO.ipSpare_3
    RoundedRectangle (18,468 25x25), colour toggle: arrTCMultiLevel[iHMICbLevelSelection].fbTCMultiLevelSeq.stMLDIO.ipSpare_4
    RoundedRectangle (18,499 25x25), colour toggle: arrTCMultiLevel[iHMICbLevelSelection].fbTCMultiLevelSeq.stMLDIO.ipCellFluidLeakage1
    RoundedRectangle (18,530 25x25), colour toggle: arrTCMultiLevel[iHMICbLevelSelection].fbTCMultiLevelSeq.stMLDIO.ipCellFluidLeakage2
    RoundedRectangle (18,561 25x25), colour toggle: arrTCMultiLevel[iHMICbLevelSelection].fbTCMultiLevelSeq.stMLDIO.ipCellGroundFault
    RoundedRectangle (18,592 25x25)
    RoundedRectangle (18,623 25x25)
    RoundedRectangle (18,654 25x25)
    RoundedRectangle (791,251 200x25), "opCellDrawerCylRetract"
        toggle arrTCMultiLevel[iHMICbLevelSelection].fbTCMultiLevelSeq.stMLDIO.opCellDrawerCylRetract
    RoundedRectangle (791,282 200x25), "opCellDrawerCylUp"
        toggle arrTCMultiLevel[iHMICbLevelSelection].fbTCMultiLevelSeq.stMLDIO.opCellDrawerCylUp
    RoundedRectangle (791,313 200x25), "opCellDrawerCylDown"
        toggle arrTCMultiLevel[iHMICbLevelSelection].fbTCMultiLevelSeq.stMLDIO.opCellDrawerCylDown
    RoundedRectangle (791,344 200x25), "opTst240VACPwrEnable"
        toggle arrTCMultiLevel[iHMICbLevelSelection].fbTCMultiLevelSeq.stMLDIO.opTst240VACPwrEnable
    RoundedRectangle (791,375 200x25), "opSpare_9"
        toggle arrTCMultiLevel[iHMICbLevelSelection].fbTCMultiLevelSeq.stMLDIO.opSpare_9
    RoundedRectangle (791,406 200x25), "opSpare_10"
        toggle arrTCMultiLevel[iHMICbLevelSelection].fbTCMultiLevelSeq.stMLDIO.opSpare_10
    RoundedRectangle (791,437 200x25), "opCellPCWValve"
        toggle arrTCMultiLevel[iHMICbLevelSelection].fbTCMultiLevelSeq.stMLDIO.opCellPCWValve
    RoundedRectangle (791,468 200x25), "opAPTIUSktCoolingAir1"
        toggle arrTCMultiLevel[iHMICbLevelSelection].fbTCMultiLevelSeq.stMLDIO.opTIUSktAirSol_1
    RoundedRectangle (791,499 200x25), "opAPTIUSktCoolingAir2"
        toggle arrTCMultiLevel[iHMICbLevelSelection].fbTCMultiLevelSeq.stMLDIO.opTIUSktAirSol_2
    RoundedRectangle (791,530 200x25), "opAPAirSupplySol"
        toggle arrTCMultiLevel[iHMICbLevelSelection].fbTCMultiLevelSeq.stMLDIO.opAPAirSupplySol
    RoundedRectangle (791,561 200x25), "opTesterDrawerAirSupplySol"
        toggle arrTCMultiLevel[iHMICbLevelSelection].fbTCMultiLevelSeq.stMLDIO.opTesterDrawerAirSupplySol
    RoundedRectangle (791,592 200x25), "opCell24VPowerEnable"
        toggle arrTCMultiLevel[iHMICbLevelSelection].fbTCMultiLevelSeq.stMLDIO.opCell24VPowerEnable
    RoundedRectangle (791,623 200x25), "opFrontDoorLock1 (DC)"
        toggle arrTCMultiLevel[iHMICbLevelSelection].fbTCMultiLevelSeq.stMLDIO.opCellTBOtSideDoorClosed1
    RoundedRectangle (791,685 200x25), "opCellDoorLock"
        toggle arrTCMultiLevel[iHMICbLevelSelection].fbTCMultiLevelSeq.stMLDIO.opCellDoorClosed
    RoundedRectangle (764,220 25x25), colour toggle: arrTCMultiLevel[iHMICbLevelSelection].fbTCMultiLevelSeq.stMLDIO.opCellDrawerCylExtend
    RoundedRectangle (764,251 25x25), colour toggle: arrTCMultiLevel[iHMICbLevelSelection].fbTCMultiLevelSeq.stMLDIO.opCellDrawerCylRetract
    RoundedRectangle (764,282 25x25), colour toggle: arrTCMultiLevel[iHMICbLevelSelection].fbTCMultiLevelSeq.stMLDIO.opCellDrawerCylUp
    RoundedRectangle (764,313 25x25), colour toggle: arrTCMultiLevel[iHMICbLevelSelection].fbTCMultiLevelSeq.stMLDIO.opCellDrawerCylDown
    RoundedRectangle (764,344 25x25), colour toggle: arrTCMultiLevel[iHMICbLevelSelection].fbTCMultiLevelSeq.stMLDIO.opTst240VACPwrEnable
    RoundedRectangle (764,375 25x25), colour toggle: arrTCMultiLevel[iHMICbLevelSelection].fbTCMultiLevelSeq.stMLDIO.opSpare_9
    RoundedRectangle (764,406 25x25), colour toggle: arrTCMultiLevel[iHMICbLevelSelection].fbTCMultiLevelSeq.stMLDIO.opSpare_10
    RoundedRectangle (764,437 25x25), colour toggle: arrTCMultiLevel[iHMICbLevelSelection].fbTCMultiLevelSeq.stMLDIO.opCellPCWValve
    RoundedRectangle (764,468 25x25), colour toggle: arrTCMultiLevel[iHMICbLevelSelection].fbTCMultiLevelSeq.stMLDIO.opTIUSktAirSol_1
    RoundedRectangle (764,499 25x25), colour toggle: arrTCMultiLevel[iHMICbLevelSelection].fbTCMultiLevelSeq.stMLDIO.opTIUSktAirSol_2
    RoundedRectangle (764,530 25x25), colour toggle: arrTCMultiLevel[iHMICbLevelSelection].fbTCMultiLevelSeq.stMLDIO.opAPAirSupplySol
    RoundedRectangle (764,561 25x25), colour toggle: arrTCMultiLevel[iHMICbLevelSelection].fbTCMultiLevelSeq.stMLDIO.opTesterDrawerAirSupplySol
    RoundedRectangle (764,592 25x25), colour toggle: arrTCMultiLevel[iHMICbLevelSelection].fbTCMultiLevelSeq.stMLDIO.opCell24VPowerEnable
    RoundedRectangle (764,623 25x25), colour toggle: arrTCMultiLevel[iHMICbLevelSelection].fbTCMultiLevelSeq.stMLDIO.opCellTBOtSideDoorClosed1
    RoundedRectangle (764,654 25x25), colour toggle: arrTCMultiLevel[iHMICbLevelSelection].fbTCMultiLevelSeq.stMLDIO.opCellTBOtSideDoorClosed2
    RoundedRectangle (764,685 25x25), colour toggle: arrTCMultiLevel[iHMICbLevelSelection].fbTCMultiLevelSeq.stMLDIO.opCellDoorClosed
    RoundedRectangle (289,220 200x25), "ipTesterPresent"
    RoundedRectangle (289,251 200x25), "ipTesterPowerOn"
    RoundedRectangle (289,282 200x25), "ipTesterReady"
    RoundedRectangle (289,313 200x25), "ipSpare_9"
    RoundedRectangle (289,344 200x25), "ipSpare_10"
    RoundedRectangle (289,375 200x25), "ipTCDrawerCylExtendRS"
    RoundedRectangle (289,406 200x25), "ipTCDrawerCylRetractRS"
    RoundedRectangle (289,437 200x25), "ipTCDrawerCylUpRS"
    RoundedRectangle (289,468 200x25), "ipTCDrawerCylDownRS"
    RoundedRectangle (289,499 200x25), "ipTCCellDoorLocked"
    RoundedRectangle (289,530 200x25), "ipTCCellDoorClosed"
    RoundedRectangle (289,561 200x25), "ipTesterLatchesClosed"
    RoundedRectangle (289,592 200x25), "ipTCCellAbortFlowBtn"
    RoundedRectangle (289,623 200x25), "ipTCCellDoorOpenReqBtn"
    RoundedRectangle (289,654 200x25), "ipTIUPresent"
    RoundedRectangle (289,685 200x25), "ipDrawerMaintenanceModeBtn"
    RoundedRectangle (262,220 25x25), colour toggle: arrTCMultiLevel[iHMICbLevelSelection].fbTCMultiLevelSeq.stMLDIO.ipTesterPresent
    RoundedRectangle (262,251 25x25), colour toggle: arrTCMultiLevel[iHMICbLevelSelection].fbTCMultiLevelSeq.stMLDIO.ipTesterPowerOn
    RoundedRectangle (262,282 25x25), colour toggle: arrTCMultiLevel[iHMICbLevelSelection].fbTCMultiLevelSeq.stMLDIO.ipTesterReady
    RoundedRectangle (262,313 25x25), colour toggle: arrTCMultiLevel[iHMICbLevelSelection].fbTCMultiLevelSeq.stMLDIO.ipSpare_9
    RoundedRectangle (262,344 25x25), colour toggle: arrTCMultiLevel[iHMICbLevelSelection].fbTCMultiLevelSeq.stMLDIO.ipSpare_10
    RoundedRectangle (262,375 25x25), colour toggle: arrTCMultiLevel[iHMICbLevelSelection].fbTCMultiLevelSeq.stMLDIO.ipTCDrawerCylExtendRS
    RoundedRectangle (262,406 25x25), colour toggle: arrTCMultiLevel[iHMICbLevelSelection].fbTCMultiLevelSeq.stMLDIO.ipTCDrawerCylRetractRS
    RoundedRectangle (262,437 25x25), colour toggle: arrTCMultiLevel[iHMICbLevelSelection].fbTCMultiLevelSeq.stMLDIO.ipTCDrawerCylUpRS
    RoundedRectangle (262,468 25x25), colour toggle: arrTCMultiLevel[iHMICbLevelSelection].fbTCMultiLevelSeq.stMLDIO.ipTCDrawerCylDownRS
    RoundedRectangle (262,499 25x25), colour toggle: arrTCMultiLevel[iHMICbLevelSelection].fbTCMultiLevelSeq.stMLDIO.ipTCCellDoorClosed
    RoundedRectangle (262,530 25x25), colour toggle: arrTCMultiLevel[iHMICbLevelSelection].fbTCMultiLevelSeq.stMLDIO.ipTCCellDoorOpenCloseStatus
    RoundedRectangle (262,561 25x25), colour toggle: arrTCMultiLevel[iHMICbLevelSelection].fbTCMultiLevelSeq.stMLDIO.ipTesterLatchesClosed
    RoundedRectangle (262,592 25x25), colour toggle: arrTCMultiLevel[iHMICbLevelSelection].fbTCMultiLevelSeq.stMLDIO.ipTCCellAbortFlowBtn
    RoundedRectangle (262,623 25x25), colour toggle: arrTCMultiLevel[iHMICbLevelSelection].fbTCMultiLevelSeq.stMLDIO.ipTCCellDoorOpenReqBtn
    RoundedRectangle (262,654 25x25)
    Checkbox (763,188 200x30), "Level 1 IO Diagnostic Mode", variable: arrTCMultiLevel[iHMICbLevelSelection].fbTCMultiLevelSeq.stMLVIO.bDiagnosticMode, input disabled if: TRUE
    GroupBox (6,9 493x155), "Column Inputs :"
    GroupBox (508,9 490x155), "Column Outputs :"
        RoundedRectangle (283,57 200x25), "Spare"
    RoundedRectangle (546,66 200x25), "opHotAirExhaustFan"
        toggle fbTCColumn.stTCColumnDIO.opHotAirExhaustFan
    RoundedRectangle (546,97 200x25), "Spare"
    RoundedRectangle (546,128 200x25), "Spare"
    RoundedRectangle (519,66 25x25), colour toggle: fbTCColumn.stTCColumnDIO.opHotAirExhaustFan
    RoundedRectangle (519,97 25x25)
    RoundedRectangle (519,128 25x25)
    RoundedRectangle (45,66 200x25), "ipColumnFluid_PCW_Leakage"
    RoundedRectangle (45,97 200x25), "ipAllTCDrawerRetractedinCell"
    RoundedRectangle (45,128 200x25), "ipTbotDoorClosedSignal"
    RoundedRectangle (18,66 25x25), colour toggle: fbTCColumn.stTCColumnDIO.ipColumnFluid_PCW_Leakage
    RoundedRectangle (18,97 25x25), colour toggle: fbTCColumn.stTCColumnDIO.ipAllTCDrawerRetractedinCell
    RoundedRectangle (18,128 25x25), colour toggle: fbTCColumn.stTCColumnDIO.ipTbotDoorClosedSignal
    RoundedRectangle (791,97 200x25), "Spare"
    RoundedRectangle (791,128 200x25), "Spare"
    RoundedRectangle (764,66 25x25)
    RoundedRectangle (764,97 25x25)
    RoundedRectangle (764,128 25x25)
    RoundedRectangle (289,66 200x25), "Spare"
    RoundedRectangle (289,97 200x25), "Spare"
    RoundedRectangle (289,128 200x25), "Spare"
    RoundedRectangle (262,66 25x25)
    RoundedRectangle (262,97 25x25)
    RoundedRectangle (262,128 25x25)
    Checkbox (763,32 200x30), "Column IO Diagnostic Mode", variable: bColIODiagnosticsMode
    RoundedRectangle (45,740 250x25), "ipFrontDoorClosed01"
    RoundedRectangle (45,771 250x25), "ipFrontDoorClosed02"
    RoundedRectangle (45,802 250x25), "ipFrontDoorLocked01"
    RoundedRectangle (45,833 250x25), "ipFrontDoorLocked02"
    RoundedRectangle (18,740 25x25), colour toggle: arrTCMultiLevel[iHMICbLevelSelection].fbTCMultiLevelSeq.stMLDIO.ipTCCellTbotSideDoorOpenCloseStatus01
    RoundedRectangle (18,771 25x25), colour toggle: arrTCMultiLevel[iHMICbLevelSelection].fbTCMultiLevelSeq.stMLDIO.ipTCCellTbotSideDoorOpenCloseStatus02
    RoundedRectangle (18,802 25x25), colour toggle: arrTCMultiLevel[iHMICbLevelSelection].fbTCMultiLevelSeq.stMLDIO.ipTCCellTbotSideDoorLocked01
    RoundedRectangle (18,833 25x25), colour toggle: arrTCMultiLevel[iHMICbLevelSelection].fbTCMultiLevelSeq.stMLDIO.ipTCCellTbotSideDoorLocked02
    GroupBox (505,748 493x119), "Debug Column EAP Signals :"
    RoundedRectangle (544,769 200x25), "ColumnPCWLeakageEAP"
    RoundedRectangle (544,800 200x25), "ColumnPCWSupplyLeakageEAP"
    RoundedRectangle (544,831 200x25), "ColumnPCWReturnLeakageEAP"
    RoundedRectangle (517,769 25x25), colour toggle: fbTCColumn.stTCColumnDIO.eapDColumnPCWLeakage
    RoundedRectangle (517,800 25x25), colour toggle: fbTCColumn.stTCColumnDIO.eapDColumnPCWSupplyLeakage
    RoundedRectangle (517,831 25x25), colour toggle: fbTCColumn.stTCColumnDIO.eapDColumnPCWReturnLeakage
    RoundedRectangle (788,769 200x25), "DS_Facility_eapShutOffAllACPower", colour toggle: DS_Facility_eapShutOffAllACPower
    RoundedRectangle (788,800 200x25), "ColumnPCWLeakageEAP"
    RoundedRectangle (788,831 200x25), "Spare"
    RoundedRectangle (761,769 25x25), colour toggle: DS_Facility_eapShutOffAllACPower
    RoundedRectangle (761,800 25x25), colour toggle: fbTCColumn.stTCColumnDIO.eapDColumnPCWLeakage2
    RoundedRectangle (761,831 25x25)
    Frame (1002,1 355x2000), invisible if: Not bEnableManualCommandTest1 AND Not bEnableManualCommandTest2
        shows HMI_ManualCommand()
    RoundedRectangle (1403,41 240x37), "240v AP Power(Output)", colour toggle: arrTCMultiLevel[iHMICbLevelSelection].fbTCMultiLevelSeq.stMLDIO.opAP240ACPwrEnable
    RoundedRectangle (1403,112 240x37), "240vTesterPower(Output)", colour toggle: arrTCMultiLevel[iHMICbLevelSelection].fbTCMultiLevelSeq.stMLDIO.opTst240VACPwrEnable
    RoundedRectangle (1403,184 240x50), "Cell PCW", colour toggle: arrTCMultiLevel[iHMICbLevelSelection].fbTCMultiLevelSeq.stMLDIO.opCellPCWValve
    Group (2440,7 225x262)
        Rectangle (0,0 215x259)
        Rectangle (0,237 215x22)
        RoundedRectangle (7,206 60x26), "Level[1]", tooltip "VIO Status", colour toggle: TC_ModuleState[1].Tester = E_State.eEnabled
        RoundedRectangle (7,177 60x26), "Level[2]", tooltip "VIO Status", colour toggle: TC_ModuleState[2].Tester= E_State.eEnabled
        RoundedRectangle (7,148 60x26), "Level[3]", tooltip "VIO Status", colour toggle: TC_ModuleState[3].Tester = E_State.eEnabled
        RoundedRectangle (7,119 60x26), "Level[4]", tooltip "VIO Status", colour toggle: TC_ModuleState[4].Tester = E_State.eEnabled
        RoundedRectangle (7,90 60x26), "Level[5]", tooltip "VIO Status", colour toggle: TC_ModuleState[5].Tester = E_State.eEnabled
        RoundedRectangle (7,61 60x26), "Level[6]", tooltip "VIO Status", colour toggle: TC_ModuleState[6].Tester = E_State.eEnabled
        Label (6,32 61x30), "Tester"
        RoundedRectangle (149,206 60x26), "Level[1]", tooltip "VIO Status", colour toggle: TC_ModuleState[1].TCSite[1].TIERII = E_State.eEnabled
        RoundedRectangle (149,177 60x26), "Level[2]", tooltip "VIO Status", colour toggle: TC_ModuleState[2].TCSite[1].TIERII = E_State.eEnabled
        RoundedRectangle (149,148 60x26), "Level[3]", tooltip "VIO Status", colour toggle: TC_ModuleState[3].TCSite[1].TIERII = E_State.eEnabled
        RoundedRectangle (149,119 60x26), "Level[4]", tooltip "VIO Status", colour toggle: TC_ModuleState[4].TCSite[1].TIERII = E_State.eEnabled
        RoundedRectangle (149,90 60x26), "Level[5]", tooltip "VIO Status", colour toggle: TC_ModuleState[5].TCSite[1].TIERII = E_State.eEnabled
        RoundedRectangle (149,61 60x26), "Level[6]", tooltip "VIO Status", colour toggle: TC_ModuleState[6].TCSite[1].TIERII = E_State.eEnabled
        Label (162,32 32x30), "TII"
        RoundedRectangle (78,207 60x26), "Level[1]", tooltip "VIO Status", colour toggle: TC_ModuleState[1].TCSite[1].TCU = E_State.eEnabled
        RoundedRectangle (78,178 60x26), "Level[2]", tooltip "VIO Status", colour toggle: TC_ModuleState[2].TCSite[1].TCU= E_State.eEnabled
        RoundedRectangle (78,149 60x26), "Level[3]", tooltip "VIO Status", colour toggle: TC_ModuleState[3].TCSite[1].TCU = E_State.eEnabled
        RoundedRectangle (78,120 60x26), "Level[4]", tooltip "VIO Status", colour toggle: TC_ModuleState[4].TCSite[1].TCU = E_State.eEnabled
        RoundedRectangle (78,91 60x26), "Level[5]", tooltip "VIO Status", colour toggle: TC_ModuleState[5].TCSite[1].TCU = E_State.eEnabled
        RoundedRectangle (78,62 60x26), "Level[6]", tooltip "VIO Status", colour toggle: TC_ModuleState[6].TCSite[1].TCU = E_State.eEnabled
        Label (87,33 43x30), "TCU"
        Label (12,232 213x30), "Green: Enable , Gray: Disable"
        Rectangle (0,1 215x32), "Enable/ Disable Status"
    ComboBoxInteger (1477,324 174x30), variable: TestManually.iBtnNo, text list: 'BtnTxtList'
    Label (1391,323 79x30), "Button:"
    Label (1393,518 80x30), "Level 6 :"
    Textfield (1479,518 150x30), "%s", text variable: TC_EPT[6].TCSite[1].TCU
    Label (1393,558 80x30), "Level 5 :"
    Textfield (1479,558 150x30), "%s", text variable: TC_EPT[5].TCSite[1].TCU
    Textfield (1479,598 150x30), "%s", text variable: TC_EPT[4].TCSite[1].TCU
    Textfield (1479,638 150x30), "%s", text variable: TC_EPT[3].TCSite[1].TCU
    Textfield (1479,678 150x30), "%s", text variable: TC_EPT[2].TCSite[1].TCU
    Textfield (1479,718 150x30), "%s", text variable: TC_EPT[1].TCSite[1].TCU
    Label (1393,598 80x29), "Level 4 :"
    Label (1393,718 80x30), "Level 1 :"
    Label (1393,678 80x30), "Level 2 :"
    Label (1393,638 80x30), "Level 3 :"
    Label (1477,464 151x37), "EPT States"
    Textfield (1640,518 150x30), "%s", text variable: arrTCMultiLevel[6].stGblParam.iProcessState
    Textfield (1640,598 150x30), "%s", text variable: arrTCMultiLevel[4].stGblParam.iProcessState
    Textfield (1640,558 150x30), "%s", text variable: arrTCMultiLevel[5].stGblParam.iProcessState
    Textfield (1640,638 150x30), "%s", text variable: arrTCMultiLevel[3].stGblParam.iProcessState
    Textfield (1640,718 150x30), "%s", text variable: arrTCMultiLevel[1].stGblParam.iProcessState
    Textfield (1640,678 150x30), "%s", text variable: arrTCMultiLevel[2].stGblParam.iProcessState
    Label (1636,465 158x37), "Process States"
    Line (1635,462) (1635,759)
    Label (1388,390 160x30), "Production Mode:"
    Textfield (1549,390 150x30), "%s", text variable: bProductionMode
END_VISUALIZATION

// ---- VISUs/SLTC_Monitor.TcVIS
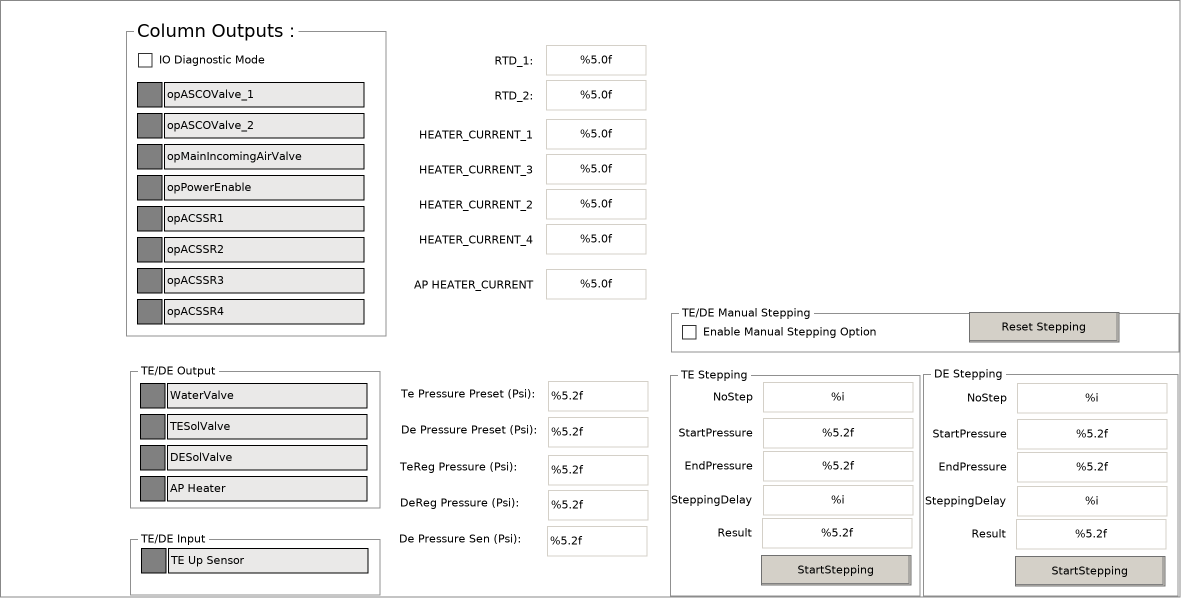
VISUALIZATION SLTC_Monitor  // 1181x598
    GroupBox (670,367 250x229), "TE Stepping"
    GroupBox (923,366 255x230), "DE Stepping"
    GroupBox (130,363 250x145), "TE/DE Output"
        RoundedRectangle (37,113 200x25), "AP Heater"
            toggle fbSLTCExtra.stDIO.opAPHeater
    GroupBox (130,531 250x64), "TE/DE Input"
    Textfield (546,45 100x30), "%5.0f", text variable: fbSLTCExtra.stVIO.ipRTD1
    Label (406,46 130x30), "RTD_1:"
    Textfield (546,80 100x30), "%5.0f", text variable: fbSLTCExtra.stVIO.ipRTD2
    Label (406,81 130x30), "RTD_2:"
    Textfield (546,119 100x30), "%5.0f", text variable: fbSLTCExtra.stVIO.ipHeaterCurrent1
    Label (406,120 130x30), "HEATER_CURRENT_1"
    Textfield (546,154 100x30), "%5.0f", text variable: fbSLTCExtra.stVIO.ipHeaterCurrent2
    Label (406,155 130x30), "HEATER_CURRENT_3"
    Textfield (546,189 100x30), "%5.0f", text variable: fbSLTCExtra.stVIO.ipHeaterCurrent3
    Label (406,190 130x30), "HEATER_CURRENT_2"
    Textfield (546,224 100x30), "%5.0f", text variable: fbSLTCExtra.stVIO.ipHeaterCurrent4
    Label (406,225 130x30), "HEATER_CURRENT_4"
    GroupBox (126,23 260x313), "Column Outputs :"
        RoundedRectangle (38,121 200x25), "opMainIncomingAirValve"
            toggle fbSLTCExtra.stDIO.opMainIncomingAirValve
        RoundedRectangle (38,183 200x25), "opACSSR1"
            toggle fbSLTCExtra.stDIO.opAC_SSR1
        RoundedRectangle (38,214 200x25), "opACSSR2"
            toggle fbSLTCExtra.stDIO.opAC_SSR2
        RoundedRectangle (11,121 25x25), colour toggle: fbSLTCExtra.stDIO.opMainIncomingAirValve
        RoundedRectangle (11,183 25x25), colour toggle: fbSLTCExtra.stDIO.opAC_SSR1
        RoundedRectangle (11,214 25x25), colour toggle: fbSLTCExtra.stDIO.opAC_SSR2
        RoundedRectangle (38,245 200x25), "opACSSR3"
            toggle fbSLTCExtra.stDIO.opAC_SSR3
        Checkbox (10,22 200x30), "IO Diagnostic Mode", variable: bColIODiagnosticsMode, invisible if: TRUE
    RoundedRectangle (164,82 200x25), "opASCOValve_1"
        toggle fbSLTCExtra.stDIO.opASCOValve_1
    RoundedRectangle (164,113 200x25), "opASCOValve_2"
        toggle fbSLTCExtra.stDIO.opASCOValve_2
    RoundedRectangle (137,82 25x25), colour toggle: fbSLTCExtra.stDIO.opASCOValve_1
    RoundedRectangle (137,113 25x25), colour toggle: fbSLTCExtra.stDIO.opASCOValve_2
    RoundedRectangle (164,299 200x25), "opACSSR4"
        toggle fbSLTCExtra.stDIO.opAC_SSR4
    RoundedRectangle (164,175 200x25), "opPowerEnable"
        toggle fbSLTCExtra.stDIO.opPowerEnable
    RoundedRectangle (137,268 25x25), colour toggle: fbSLTCExtra.stDIO.opAC_SSR3
    RoundedRectangle (137,299 25x25), colour toggle: fbSLTCExtra.stDIO.opAC_SSR4
    RoundedRectangle (137,175 25x25), colour toggle: fbSLTCExtra.stDIO.opPowerEnable
    RoundedRectangle (140,383 25x25), colour toggle: fbSLTCExtra.stDIO.opWaterValve
    RoundedRectangle (167,414 200x25), "TESolValve"
        toggle fbSLTCExtra.stDIO.opTESolValve
    RoundedRectangle (167,445 200x25), "DESolValve"
        toggle fbSLTCExtra.stDIO.opDESolValve
    RoundedRectangle (140,414 25x25), colour toggle: fbSLTCExtra.stDIO.opTESolValve
    RoundedRectangle (140,445 25x25), colour toggle: fbSLTCExtra.stDIO.opDESolValve
    RoundedRectangle (167,383 200x25), "WaterValve"
        toggle fbSLTCExtra.stDIO.opWaterValve
    RoundedRectangle (141,548 25x25), colour toggle: fbSLTCExtra.stDIO.ipTEUpRS
    RoundedRectangle (168,548 200x25), "TE Up Sensor"
    Textfield (548,381 100x30), "%5.2f", text variable: fbSLTCExtra.stVIO.opTEPressRegAOut, input disabled if: fbSLTCExtra.isEnManStepping
        OnMouseDown: write the text variable via Default, min 0, max 130
    Label (398,379 135x30), "Te Pressure Preset (Psi):"
    Textfield (548,417 100x30), "%5.2f", text variable: fbSLTCExtra.stVIO.opDEPressRegAOut
        OnMouseClick: write the text variable via Default, min 0, max 130
    Label (398,415 135x30), "De Pressure Preset (Psi):"
    Label (397,452 125x30), "TeReg Pressure (Psi):"
    Textfield (548,490 100x30), "%5.2f", text variable: fbSLTCExtra.stVIO.ipDEPressRegFeedBack
    Label (397,488 125x30), "DeReg Pressure (Psi):"
    Textfield (548,455 100x30), "%5.2f", text variable: fbSLTCExtra.stVIO.ipTEPressRegFeedBack
    Textfield (547,526 100x30), "%5.2f", text variable: fbSLTCExtra.stVIO.ipDEPressureSensor
    Label (396,524 125x30), "De Pressure Sen (Psi):"
    Textfield (763,382 150x30), "%i", text variable: fbSLTCExtra.noOfStepTE, input disabled if: Not fbSLTCExtra.isEnManStepping
        OnMouseClick: write the text variable via Default
    Label (666,382 90x30), "NoStep"
    Button (761,555 150x30), "StartStepping", input disabled if: fbSLTCExtra.isStartSteppingTE OR Not fbSLTCExtra.isEnManStepping
        tap fbSLTCExtra.btnToggleTE p1329445385=TRUE
    Textfield (763,418 150x30), "%5.2f", text variable: fbSLTCExtra.startPressureTE, input disabled if: Not fbSLTCExtra.isEnManStepping
        OnMouseClick: write the text variable via Default
    Label (666,418 90x30), "StartPressure"
    Textfield (763,451 150x30), "%5.2f", text variable: fbSLTCExtra.endPressureTE, input disabled if: Not fbSLTCExtra.isEnManStepping
        OnMouseClick: write the text variable via Default
    Label (666,451 90x30), "EndPressure"
    Textfield (763,485 150x30), "%i", text variable: fbSLTCExtra.StepDelayTE, input disabled if: Not fbSLTCExtra.isEnManStepping
        OnMouseClick: write the text variable via Default
    Label (665,485 90x30), "SteppingDelay"
    Label (665,518 90x30), "Result"
    Textfield (762,518 150x30), "%5.2f", text variable: fbSLTCExtra.TEResult, input disabled if: TRUE
    Checkbox (680,317 215x30), "Enable Manual Stepping Option", variable: fbSLTCExtra.isEnManStepping
    Textfield (1017,383 150x30), "%i", text variable: fbSLTCExtra.noOfStepDE, input disabled if: Not fbSLTCExtra.isEnManStepping
        OnMouseClick: write the text variable via Default
    Label (920,383 90x30), "NoStep"
    Button (1015,556 150x30), "StartStepping", input disabled if: fbSLTCExtra.isStartSteppingDE OR Not fbSLTCExtra.isEnManStepping
        tap fbSLTCExtra.btnToggleDE p1329445385=TRUE
    Textfield (1017,419 150x30), "%5.2f", text variable: fbSLTCExtra.startPressureDE, input disabled if: Not fbSLTCExtra.isEnManStepping
        OnMouseClick: write the text variable via Default
    Label (920,419 90x30), "StartPressure"
    Textfield (1017,452 150x30), "%5.2f", text variable: fbSLTCExtra.endPressureDE, input disabled if: Not fbSLTCExtra.isEnManStepping
        OnMouseClick: write the text variable via Default
    Label (920,452 90x30), "EndPressure"
    Textfield (1017,486 150x30), "%i", text variable: fbSLTCExtra.StepDelayDE, input disabled if: Not fbSLTCExtra.isEnManStepping
        OnMouseClick: write the text variable via Default
    Label (919,486 90x30), "SteppingDelay"
    Label (919,519 90x30), "Result"
    Textfield (1016,519 150x30), "%5.2f", text variable: fbSLTCExtra.DEResult, input disabled if: TRUE
    GroupBox (671,305 508x47), "TE/DE Manual Stepping"
        Button (298,7 150x30), "Reset Stepping", input disabled if: fbSLTCExtra.isStartSteppingTE AND fbSLTCExtra.isStartSteppingDE OR Not fbSLTCExtra.isEnManStepping
            tap fbSLTCExtra.isResetStepping
    RoundedRectangle (140,476 25x25), colour toggle: fbSLTCExtra.stDIO.opAPHeater
    Textfield (546,269 100x30), "%5.0f", text variable: fbSLTCExtra.stVIO.ipAPHeaterCurrent
    Label (388,270 148x30), "AP HEATER_CURRENT"
END_VISUALIZATION

// ---- VISUs/Template/AIN_Template.TcVIS
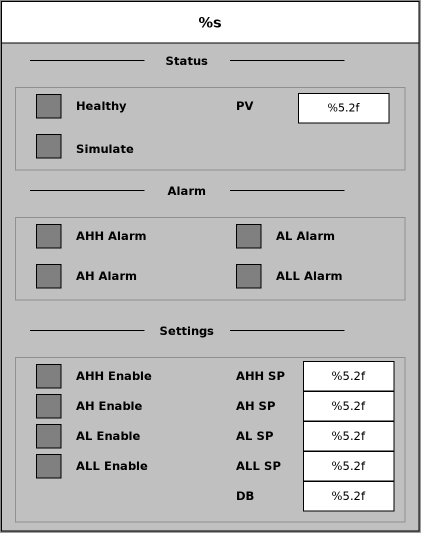
VISUALIZATION AIN_Template  // 421x533
VAR_IN_OUT
	DUT								: DUT_AIN;
END_VAR
    Group (1,1 418x530)
        Rectangle (0,0 418x530)
        Rectangle (0,0 418x42)
    Textfield (1,4 418x37), "%s", text variable: DUT.AIN_ID
    Line (30,330) (144,330)
    Line (230,330) (344,330)
    GroupBox (15,349 390x173)
        RoundedRectangle (21,45 25x24), colour toggle: DUT.AH_Enable
            toggle DUT.AH_Enable
        RoundedRectangle (21,75 25x24), colour toggle: DUT.AL_Enable
            toggle DUT.AL_Enable
        RoundedRectangle (21,105 25x24), colour toggle: DUT.ALL_Enable
            toggle DUT.ALL_Enable
        Label (218,42 64x30), "AH SP"
        Label (218,72 64x30), "AL SP"
        Label (218,102 64x30), "ALL SP"
        Label (218,132 64x30), "DB"
    RoundedRectangle (36,364 25x24), colour toggle: DUT.AHH_Enable
        toggle DUT.AHH_Enable
    Label (73,361 100x30), "AHH Enable"
    Label (233,361 64x30), "AHH SP"
    Label (112,316 150x30), "Settings"
    Label (73,391 100x30), "AH Enable"
    Label (73,421 100x30), "AL Enable"
    Label (73,451 100x30), "ALL Enable"
    Rectangle (303,361 91x30), "%5.2f", text variable: DUT.AHH_SP
        OnMouseClick: write DUT.AHH_SP via Default
    Rectangle (303,391 91x30), "%5.2f", text variable: DUT.AH_SP
        OnMouseClick: write DUT.AH_SP via Default
    Rectangle (303,421 91x30), "%5.2f", text variable: DUT.AL_SP
        OnMouseClick: write DUT.AL_SP via Default
    Rectangle (303,451 91x30), "%5.2f", text variable: DUT.ALL_SP
        OnMouseClick: write DUT.ALL_SP via Default
    Rectangle (303,481 91x30), "%5.2f", text variable: DUT.DB
        OnMouseClick: write DUT.DB via Default
    Line (30,60) (144,60)
    Line (230,60) (344,60)
    GroupBox (15,79 390x91)
        Label (218,12 64x30), "PV"
        Rectangle (283,14 91x30), "%5.2f", text variable: DUT.PV
            OnMouseClick: write DUT.PV via Default
    RoundedRectangle (36,94 25x24), colour toggle: DUT.Healthy
    Label (73,91 64x30), "Healthy"
    Label (73,134 64x30), "Simulate"
    RoundedRectangle (36,134 25x24), colour toggle: DUT.Simulate
        toggle DUT.Simulate
    Label (112,46 150x30), "Status"
    Line (30,190) (144,190)
    Line (230,190) (344,190)
    GroupBox (15,209 390x91)
        RoundedRectangle (21,55 25x24), colour toggle: DUT.AH
        RoundedRectangle (221,55 25x24), colour toggle: DUT.ALL
    RoundedRectangle (36,224 25x24), colour toggle: DUT.AHH
    Label (73,221 100x30), "AHH Alarm"
    Label (112,176 150x30), "Alarm"
    Label (73,261 100x30), "AH Alarm"
    RoundedRectangle (236,224 25x24), colour toggle: DUT.AL
    Label (273,221 100x30), "AL Alarm"
    Label (273,261 100x30), "ALL Alarm"
END_VISUALIZATION

// ---- VISUs/Template/Cylinder_Template.TcVIS
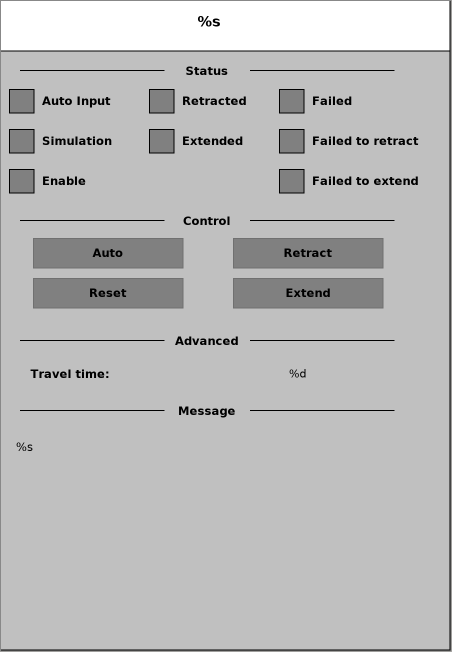
VISUALIZATION Cylinder_Template  // 452x652
VAR_IN_OUT
	DUT										: DUT_Cylinder;
END_VAR
    Group (0,0 418x530)
        Rectangle (0,0 450x650)
        Rectangle (0,0 450x51)
    Label (132,56 150x30), "Status"
    Line (20,70) (164,70)
    Label (132,206 150x30), "Control"
    Label (132,326 150x30), "Advanced"
    Label (132,396 150x30), "Message"
    Textfield (0,3 418x37), "%s", text variable: DUT.CylinderID
    RoundedRectangle (9,89 25x24), colour toggle: DUT.AutInp
    Label (39,86 106x30), "Auto Input"
    Label (39,126 106x30), "Simulation"
    RoundedRectangle (9,129 25x24), colour toggle: DUT.Simulate
    Label (39,166 106x30), "Enable"
    RoundedRectangle (9,169 25x24), colour toggle: DUT.Enable
    RoundedRectangle (279,89 25x24), colour toggle: DUT.Failed
    Label (309,86 106x30), "Failed"
    Label (309,126 106x30), "Failed to retract"
    RoundedRectangle (279,129 25x24), colour toggle: DUT.Failed_To_Retract
    Label (309,166 106x30), "Failed to extend"
    RoundedRectangle (279,169 25x24), colour toggle: DUT.Failed_To_Extend
    Button (33,238 150x30), "Auto", colour toggle: DUT.CMD = 4
        OnMouseClick: execute { DUT.CMD			:= 4; }
    Button (33,278 150x30), "Reset", colour toggle: DUT.Reset
        toggle DUT.Reset
    Button (233,238 150x30), "Retract", colour toggle: DUT.CMD = 1
        OnMouseClick: execute { DUT.CMD			:= 1; }
    Button (233,278 150x30), "Extend", colour toggle: DUT.CMD = 2
        OnMouseClick: execute { DUT.CMD			:= 2; }
    Label (16,359 108x30), "Travel time:"
    Textfield (223,359 150x30), "%d", text variable: DUT.Travel_Time
        OnMouseClick: write DUT.Travel_Time via Default, min 1, max 999
    Textfield (13,439 392x76), "%s", text variable: DUT.Message
    Line (250,70) (394,70)
    Line (250,220) (394,220)
    Line (20,220) (164,220)
    Line (250,340) (394,340)
    Line (20,340) (164,340)
    Line (250,410) (394,410)
    Line (20,410) (164,410)
    RoundedRectangle (149,89 25x24), colour toggle: DUT.Retracted
    Label (179,86 106x30), "Retracted"
    Label (179,126 106x30), "Extended"
    RoundedRectangle (149,129 25x24), colour toggle: DUT.Extended
END_VISUALIZATION
